FUNCTION_BLOCK SPLIT_AB_INTO_AQ (* this Function splits the 4 AQ (QUARTER) adapters from a AB (BYTE) *)
  (* Standard: 61499-2; Description: Copyright (c) 2026 Meisterschulen am Ostbahnhof SPDX-License-Identifier: EPL-2.0 *)
  (* Version 1.0, 2026-05-16, Franz Höpfinger, Meisterschulen am Ostbahnhof, initial API and implementation and/or initial documentation *)
  PACKAGE adapter::splitting;
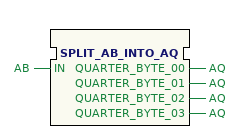
  SOCKETS
    IN : adapter::types::unidirectional::AB; (* BYTE Input *)
  END_SOCKETS
  PLUGS
    QUARTER_BYTE_00 : adapter::types::unidirectional::AQ; (* Quarter 0 *)
    QUARTER_BYTE_01 : adapter::types::unidirectional::AQ; (* Quarter 1 *)
    QUARTER_BYTE_02 : adapter::types::unidirectional::AQ; (* Quarter 2 *)
    QUARTER_BYTE_03 : adapter::types::unidirectional::AQ; (* Quarter 3 *)
  END_PLUGS
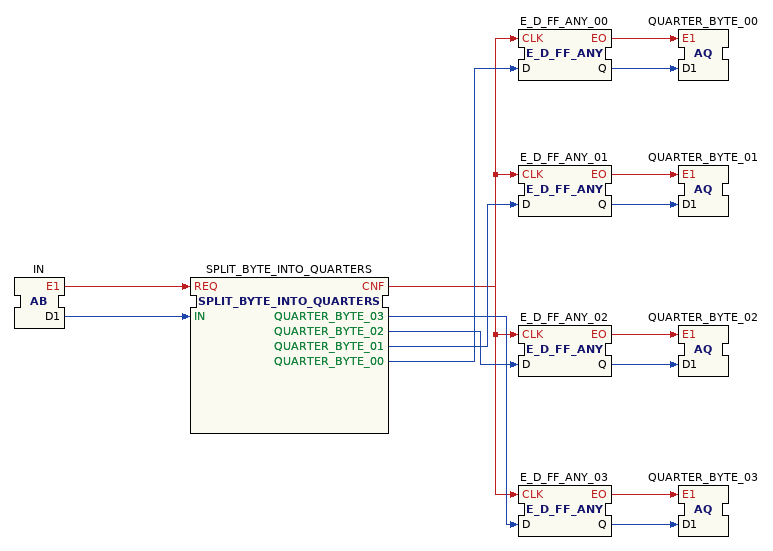
  FBS
    E_D_FF_ANY_00 : iec61499::events::E_D_FF_ANY;
    E_D_FF_ANY_01 : iec61499::events::E_D_FF_ANY;
    E_D_FF_ANY_02 : iec61499::events::E_D_FF_ANY;
    E_D_FF_ANY_03 : iec61499::events::E_D_FF_ANY;
    SPLIT_BYTE_INTO_QUARTERS : eclipse4diac::utils::splitting::SPLIT_BYTE_INTO_QUARTERS;
  END_FBS
  EVENT_CONNECTIONS
    IN.E1 TO SPLIT_BYTE_INTO_QUARTERS.REQ;
    SPLIT_BYTE_INTO_QUARTERS.CNF TO E_D_FF_ANY_00.CLK;
    SPLIT_BYTE_INTO_QUARTERS.CNF TO E_D_FF_ANY_01.CLK;
    SPLIT_BYTE_INTO_QUARTERS.CNF TO E_D_FF_ANY_02.CLK;
    SPLIT_BYTE_INTO_QUARTERS.CNF TO E_D_FF_ANY_03.CLK;
    E_D_FF_ANY_00.EO TO QUARTER_BYTE_00.E1;
    E_D_FF_ANY_01.EO TO QUARTER_BYTE_01.E1;
    E_D_FF_ANY_02.EO TO QUARTER_BYTE_02.E1;
    E_D_FF_ANY_03.EO TO QUARTER_BYTE_03.E1;
  END_CONNECTIONS
  DATA_CONNECTIONS
    IN.D1 TO SPLIT_BYTE_INTO_QUARTERS.IN;
    SPLIT_BYTE_INTO_QUARTERS.QUARTER_BYTE_03 TO E_D_FF_ANY_03.D;
    SPLIT_BYTE_INTO_QUARTERS.QUARTER_BYTE_02 TO E_D_FF_ANY_02.D;
    SPLIT_BYTE_INTO_QUARTERS.QUARTER_BYTE_01 TO E_D_FF_ANY_01.D;
    SPLIT_BYTE_INTO_QUARTERS.QUARTER_BYTE_00 TO E_D_FF_ANY_00.D;
    E_D_FF_ANY_00.Q TO QUARTER_BYTE_00.D1;
    E_D_FF_ANY_01.Q TO QUARTER_BYTE_01.D1;
    E_D_FF_ANY_02.Q TO QUARTER_BYTE_02.D1;
    E_D_FF_ANY_03.Q TO QUARTER_BYTE_03.D1;
  END_CONNECTIONS
END_FUNCTION_BLOCK
